(* IEC 61131-3 sources: AXOpen/src/components.elements/ctrl/src/AxoAi, 3 files *)

(* ---- AxoAi.st ---- *)
USING AXOpen.Core;
NAMESPACE AXOpen.Components.Elements
    /// <summary>
    /// Class representing Analog input
    /// </summary>
    {S7.extern=ReadWrite}
    CLASS AxoAi EXTENDS AXOpen.Core.AxoComponent

        VAR PUBLIC
            /// configuration for calculations
            {#ix-attr:[Container(Layout.Wrap)]}
            {#ix-attr:[ComponentDetails("Config")]}
            _config : AxoAiConfig;

            /// status of input
            {#ix-attr:[ComponentHeader()]}
            {#ix-attr:[Container(Layout.Wrap)]}
            {#ix-attr:[Group(GroupLayout.GroupBox)]}
            {#ix-attr:[ReadOnly()]}
            {#ix-set:AttributeName = "<#Status#>"}
            _status : AxoAiStatus;

            {#ix-attr:[Container(Layout.Wrap)]}
            _rawRange : REAL;
            _realRange : REAL;
            _scaled : REAL;

            {#ix-set:AttributeName = "<#MessengerInfo#>"}
            {#ix-set:PlcTextList = "[1]:'<#Division by zero: Verify values defined in config! (RawHigh,RawLow)':'<#Check the scaling parameters.#>';[2]:'<#Invalid data: Gain is not defined!#>':'<#Check the scaling parameters.#>';[3]:'<#Out of boundaries,check correction parameters (Gain,Ofset) in config!#>':'<#Check your signal input.#>'"}
            _messengerInfo : AXOpen.Messaging.Static.AxoMessenger;
        END_VAR

        VAR
            _signal : DINT;
        END_VAR

        VAR PRIVATE
            _context : IAxoContext;
        END_VAR

        /// <summary>
        /// Method, which scales input signal based on configuration
        /// </summary>
        METHOD PUBLIC Run

            VAR_INPUT
                parent : Axopen.Core.IAxoObject;
                inSignal: DINT;
            END_VAR

            IF (parent = NULL) THEN
                RETURN;
            END_IF;

            IF _context = NULL THEN
                SUPER.Run(parent);
                _context := THIS.GetContext();
            END_IF;

            _messengerInfo.Serve(THIS);

            _signal := inSignal;
            //scaling
            _rawRange  := TO_REAL(_config.RawHigh - _config.RawLow);
            _realRange := _config.RealHigh - _config.RealLow;
            _scaled    := 0;

            IF (_rawRange = 0) THEN
                _messengerInfo.Activate(UINT#1,AXOpen.Messaging.eAxoMessageCategory#Error);
                RETURN;
            END_IF;

            IF (_config.Gain = 0) THEN
                _messengerInfo.Activate(UINT#2,AXOpen.Messaging.eAxoMessageCategory#Error);
            END_IF;

            _scaled := TO_REAL(_signal - _config.RawLow) / _rawRange;

            _scaled := _scaled * _realRange;
            _scaled := _scaled + _config.RealLow;

            _scaled := _scaled * _config.Gain + _config.Offset;

            IF (_scaled > _config.RealHigh) AND (_config.Gain <> 1 OR _config.Offset <> 0) THEN
                _messengerInfo.Activate(UINT#3,AXOpen.Messaging.eAxoMessageCategory#Error);
            ELSIF (_scaled < _config.RealLow) AND (_config.Gain <> 1 OR _config.Offset <> 0) THEN
                _messengerInfo.Activate(UINT#3,AXOpen.Messaging.eAxoMessageCategory#Error);
            END_IF;

            _status.RawRange  := _rawRange;
            _status.RealRange := _realRange;
            _status.Scaled    := _scaled;
        END_METHOD

        /// <summary>
        /// Method, which scales input signal based on configuration
        /// </summary>
        METHOD PUBLIC Run
            VAR_INPUT
                parent : Axopen.Core.IAxoObject;
                inSignal: WORD;
            END_VAR
            THIS.Run(parent,TO_DINT(inSignal));
        END_METHOD

        METHOD PUBLIC OVERRIDE Restore
            ;
        END_METHOD

        METHOD PROTECTED OVERRIDE ManualControl
            THIS._isManuallyControllable := TRUE;
        END_METHOD
    END_CLASS
END_NAMESPACE

(* ---- AxoAiConfig.st ---- *)
NAMESPACE AXOpen.Components.Elements
    // <AxoAiConfigDeclaration>
    // <summary>
    // Configuration class for analog input
    // </summary>
    {S7.extern=ReadWrite}
    CLASS AxoAiConfig
        VAR PUBLIC

        // <summary>
        // Lowest possible value of the raw input.
        // </summary>
        RawLow : DINT;

        // <summary>
        // Highest possible value of the raw input.
        // </summary>
        RawHigh : DINT;

        // <summary>
        // Lowest threshold of scaled value.
        // `RealLow` and `RealHigh` should represent the real range of an continuous input.
        // </summary>
        RealLow  : REAL;

        // <summary>
        // Highest threshold range of scaled value.
        // `RealLow` and `RealHigh` should represent the real range of an continuous input.
        // </summary>
        RealHigh : REAL;

		// <summary>
		// Allows simple adjustment of the calculated value multiplying the value by factor of `Gain`.
		// </summary>
        Gain : REAL := REAL#1.0;
        // <summary>
        // Allows simple adjustment of the calculated value by adding `Offset` value.
        // </summary>
        Offset : REAL := REAL#0.0;
        END_VAR
    END_CLASS
    // </AxoAiConfigDeclaration>
END_NAMESPACE

(* ---- AxoAiStatus.st ---- *)
NAMESPACE AXOpen.Components.Elements

    /// <summary>
    /// 	Class representing current status of analog input
    /// </summary>
    {S7.extern=ReadWrite}
    CLASS AxoAiStatus
        VAR PUBLIC
        // <summary>
        // 	Absolute range of raw value.
        // </summary>
        {#ix-set:AttributeName = "<#Raw range#>"}
        RawRange : REAL;

        // <summary>
        // 	Absolute range of real value.
        // </summary>
        {#ix-set:AttributeName = "<#Real range#>"}
        RealRange : REAL;
        // <summary>
        // Current real value.
        // </summary>
        {#ix-set:AttributeName = "<#Scale value#>"}
        Scaled : REAL;
        END_VAR
    END_CLASS
END_NAMESPACE
